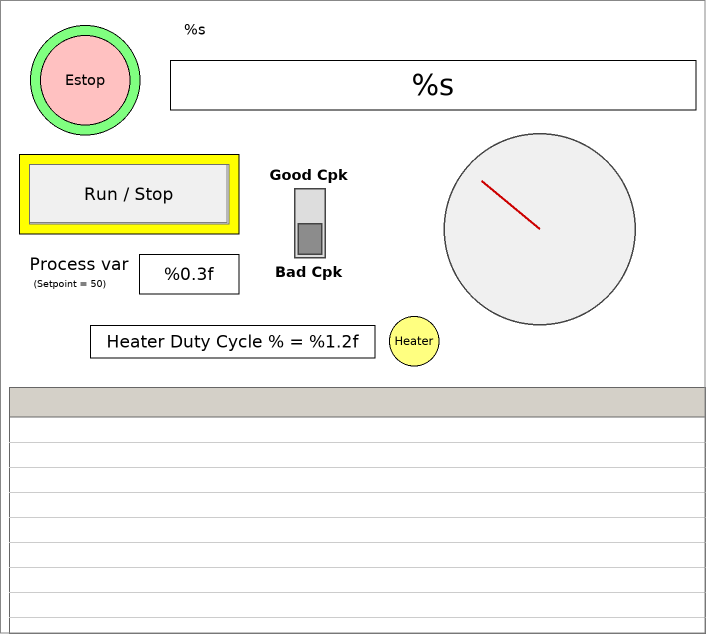
VISUALIZATION Visualization  // 706x634
    Rectangle (265,158 87x34), "Good Cpk"
    Ellipse (30,25 110x110), colour toggle: MAIN.bEstop
    Ellipse (40,35 90x90), "Estop"
        toggle MAIN.bEstop
    Rectangle (170,60 526x50), "%s", text variable: MAIN.sState
    Rectangle (181,17 255x25), "%s", text variable: MAIN.sDateTimeLocal
    Rectangle (19,154 220x80), colour toggle: MAIN.bRun
    Button (29,164 200x60), "Run / Stop", pressed state: MAIN.bRun
        toggle MAIN.bRun
    Rectangle (139,254 100x40), "%0.3f", text variable: MAIN.rRealVal
        OnMouseDown: write the text variable via VisuDialogs.Keypad
    Rectangle (14,249 130x30), "Process var"
    Rectangle (34,269 75x30), "(Setpoint = 50)"
    Meter180 (375,133 329x192), value: MAIN.rRealVal, style: Meter-Meter180-Gray, scale format: %.1f, scale 0..100
    Rectangle (90,325 285x33), "Heater Duty Cycle % = %1.2f", text variable: MAIN.rDutyCycle
        OnMouseDown: write the text variable via VisuDialogs.Numpad, min 1, max 100
    Ellipse (389,316 50x50), "Heater", colour toggle: MAIN.bHeater
    Table (9,387 697x247), data array: MAIN.stEventArray
        p3854506369: MAIN.stEventArray[INDEX].sDateTime
        p1892666644: MAIN.stEventArray[INDEX].sEvent
        p338671338: MAIN.stEventArray[INDEX].fProcVal
        p1755163831: Process Value
        p1128707560: MAIN.iNumEvents
        p2170511999: MAIN.stEventArray[INDEX].bHeaterState
        p4092479075: Heater State
    Rectangle (265,255 87x34), "Bad Cpk"
    DipSwitch (275,188 70x70), variable: MAIN.bGoodCpk, behaviour: TOGGLE, style: Switch-DipSwitch-Gray
END_VISUALIZATION

(* stored: Version 1.1.0.1, ProductVersion 3.1.4024.4
   Visu Visualization: Id {906589f6-b989-4f71-8545-61ecc4b40da4} *)
